// TIA Portal V15.1 export
// export: Created 2019-08-14T06:24:31.9270763Z, ExportSetting None, DisplayName Totally Integrated Automation Portal, DisplayVersion V15.1, DisplayName TIA Portal Openness, DisplayVersion V15.1, DisplayName STEP 7 Professional, DisplayVersion V15.1, DisplayName STEP 7 Safety, DisplayVersion V15.1, DisplayName WinCC Advanced, DisplayVersion V15.1
DATA_BLOCK "SkillStateMachineMapping"   // DB5
{ S7_Optimized_Access := 'TRUE' }
// stored: InstanceOfName typeSkillStateMachineMapping, InstanceOfType UDT
"typeSkillStateMachineMapping"
   // VAR
   //    SkillStateMachine : Struct
   //       CurrentState_Id : OPC_UA_NodeId;
   //       LastTransition_Id : OPC_UA_NodeId;
   //       AvailableStates_NodeIds : Array[0..2] of OPC_UA_NodeId;
   //       AvailableStates_Names : Array[0..2] of String;
   //       AvailableStates_Numbers : Array[0..2] of Byte;
   //       AvailableTransitions_NodeIds : Array[0..2] of OPC_UA_NodeId;
   //       AvailableTransitions_Names : Array[0..2] of String;
   //       AvailableTransitions_Numbers : Array[0..2] of Byte;
   //    END_STRUCT;
   //    ClearedStatMachine : Struct
   //       CurrentState_Id : OPC_UA_NodeId;
   //       LastTransition_Id : OPC_UA_NodeId;
   //       AvailableStates_NodeIds : Array[0..3] of OPC_UA_NodeId;
   //       AvailableStates_Names : Array[0..3] of String;
   //       AvailableStates_Numbers : Array[0..3] of Byte;
   //       AvailableTransitions_NodeIds : Array[0..3] of OPC_UA_NodeId;
   //       AvailableTransitions_Names : Array[0..3] of String;
   //       AvailableTransitions_Numbers : Array[0..3] of Byte;
   //    END_STRUCT;
   //    RunningStateMachine : Struct
   //       CurrentState_Id : OPC_UA_NodeId;
   //       LastTransition_Id : OPC_UA_NodeId;
   //       AvailableStates_NodeIds : Array[0..5] of OPC_UA_NodeId;
   //       AvailableStates_Names : Array[0..5] of String;
   //       AvailableStates_Numbers : Array[0..5] of Byte;
   //       AvailableTransitions_NodeIds : Array[0..6] of OPC_UA_NodeId;
   //       AvailableTransitions_Names : Array[0..6] of String;
   //       AvailableTransitions_Numbers : Array[0..6] of Byte;
   //    END_STRUCT;
   //    IdleStateMachine : Struct
   //       CurrentState_Id : OPC_UA_NodeId;
   //       LastTransition_Id : OPC_UA_NodeId;
   //       AvailableStates_NodeIds : Array[0..1] of OPC_UA_NodeId;
   //       AvailableStates_Names : Array[0..1] of String;
   //       AvailableStates_Numbers : Array[0..1] of Byte;
   //       AvailableTransitions_NodeIds : Array[0..0] of OPC_UA_NodeId;
   //       AvailableTransitions_Names : Array[0..0] of String;
   //       AvailableTransitions_Numbers : Array[0..0] of Byte;
   //    END_STRUCT;
   //    HoldStateMachine : Struct
   //       CurrentState_Id : OPC_UA_NodeId;
   //       LastTransition_Id : OPC_UA_NodeId;
   //       AvailableStates_NodeIds : Array[0..2] of OPC_UA_NodeId;
   //       AvailableStates_Names : Array[0..2] of String;
   //       AvailableStates_Numbers : Array[0..2] of Byte;
   //       AvailableTransitions_NodeIds : Array[0..1] of OPC_UA_NodeId;
   //       AvailableTransitions_Names : Array[0..1] of String;
   //       AvailableTransitions_Numbers : Array[0..1] of Byte;
   //    END_STRUCT;
   //    ResettingStateMachine : Struct
   //       CurrentState_Id : OPC_UA_NodeId;
   //       LastTransition_Id : OPC_UA_NodeId;
   //       AvailableStates_NodeIds : Array[0..2] of OPC_UA_NodeId;
   //       AvailableStates_Names : Array[0..2] of String;
   //       AvailableStates_Numbers : Array[0..2] of Byte;
   //       AvailableTransitions_NodeIds : Array[0..2] of OPC_UA_NodeId;
   //       AvailableTransitions_Names : Array[0..2] of String;
   //       AvailableTransitions_Numbers : Array[0..2] of Byte;
   //    END_STRUCT;
   //    ExecuteStateMachine : Struct
   //       CurrentState_Id : OPC_UA_NodeId;
   //       LastTransition_Id : OPC_UA_NodeId;
   //       AvailableStates_NodeIds : Array[0..1] of OPC_UA_NodeId;
   //       AvailableStates_Names : Array[0..1] of String;
   //       AvailableStates_Numbers : Array[0..1] of Byte;
   //       AvailableTransitions_NodeIds : Array[0..1] of OPC_UA_NodeId;
   //       AvailableTransitions_Names : Array[0..1] of String;
   //       AvailableTransitions_Numbers : Array[0..1] of Byte;
   //    END_STRUCT;
   // END_VAR
BEGIN
END_DATA_BLOCK
